FUNCTION_BLOCK FB_Timer
VAR_INPUT
	bStart:BOOL;
	bPause:BOOL;
	bReset:BOOL;
	Starting: BOOL;
	Running: BOOL:=FALSE;
	
END_VAR
VAR_OUTPUT
	ElapsedTime:TIME:=T#0MS;
	
END_VAR
VAR
	bStartD: R_TRIG;
	
	
END_VAR

bStartD(CLK:=bStart);
IF bStartD.Q THEN
	Starting:=TRUE;
END_IF
IF bStart AND NOT Running THEN
	Running:=True;
	bStart:=FALSE;
		
ELSIF bReset THEN
	ElapsedTime:=T#0MS;
	bReset:=FALSE;	
	Running:=FALSE;
	
	
ELSIF bPause THEN
	Running:=FALSE;
	bPause:=FALSE;

END_IF
IF Running THEN 
	ElapsedTime:=Elapsedtime+T#10ms;
END_IF

END_FUNCTION_BLOCK

(* stored: Version 1.1.0.1, ProductVersion 3.1.4026.8
   POU FB_Timer: Id {4dc440aa-a682-45de-a438-729f7294ffb8}, SpecialFunc None *)
